(* IEC 61131-3 sources: Lasal/CPU_5344_V01/Class/CanDriverCPU, 1 file *)

(* ---- CanDriverCPU.st ---- *)
(*!
<Class
	Name               = "CanDriverCPU"
	Revision           = "0.3"
	RealtimeTask       = "false"
	CyclicTask         = "false"
	BackgroundTask     = "false"
	Sigmatek           = "false"
	OSInterface        = "false"
	HighPriority       = "false"
	Automatic          = "false"
	UpdateMode         = "Prescan"
	SharedCommandTable = "true"
	Objectsize         = "(332,120)">
	<Channels>
		<Client Name="_CanLib0" Required="true" Internal="true"/>
	</Channels>
	<RevDoku>
		<Owner Company="SigmaContol" Author="Johan Embregts"/>
		<Dokumentation Revision="0.3" Date="2014-02-03" Author="Johan Embregts" Company="SigmaContol" Description="Adapted to new Revision of &quot;CanDriverBase&quot; Rev 1.0 or higher."/>
	</RevDoku>
	<Network Name="CanDriverCPU">
		<!-- List of Components in this network -->
		<Components>
			<Object
				Name       = "_base"
				Class      = "CanDriverBase"
				Position   = "(570,120)"
				Visualized = "true">
				<Channels>
					<Server Name="CobId"/>
					<Server Name="Command"/>
					<Server Name="ErrCntr"/>
					<Server Name="Status"/>
					<Client Name="CanChannel"/>
					<Client Name="cBaudrate"/>
					<Client Name="HwSelector" Value="CanDriverBase::CAN_conv"/>
					<Client Name="IrqChannel"/>
				</Channels>
			</Object>
			<Object
				Name       = "_CanLib0"
				Class      = "_CanLib"
				Position   = "(180,120)"
				Visualized = "true">
				<Channels>
					<Server Name="CanBus" Value="1"/>
					<Server Name="Command"/>
					<Client Name="To_Can"/>
				</Channels>
			</Object>
		</Components>
		<Comments>
		</Comments>
		<!-- List of Connections in this network -->
		<Connections>
			<Connection Source="_base.CanChannel" Destination="_CanLib0.Command" Vertices="(570,210),(510,210),"/>
			<Connection Source="_base.cBaudrate" Destination="this.cBaudrate" Vertices="(570,270),(38,210),"/>
			<Connection Source="_base.IrqChannel" Destination="this.IrqChannel" Vertices="(570,390),(38,270),"/>
			<Connection Source="this.Command" Destination="_base.Command" Vertices="(1042,210),(870,210),"/>
			<Connection Source="this.Status" Destination="_base.Status" Vertices="(1042,270),(870,330),"/>
			<Connection Source="this._CanLib0" Destination="_CanLib0.Command"/>
		</Connections>
		<!-- Headerfiles -->
		<Options>
		</Options>
	</Network>
</Class>
*)
#pragma using CanDriverBase

CanDriverCPU : CLASS
: CanDriverBase
  //Servers:
  //Clients:
	_CanLib0 	: CltChCmd__CanLib;
  //Variables:
  //Functions:
  //Tables:
	FUNCTION @STD
		VAR_OUTPUT
			ret_code	: CONFSTATES;
		END_VAR;
	FUNCTION GLOBAL TAB @CT_;
END_CLASS;

#pragma using _CanLib
